FUNCTION_BLOCK FbFiveRung
VAR_INPUT
	xFromSeqLogic: BOOL;
	xEStopOK: BOOL;
	xAutoMode: BOOL;
	xManMode: BOOL;
	xPushButton: BOOL;
	xSensor: BOOL;
	xResetFault: BOOL;
END_VAR
VAR_OUTPUT
	xTrigger: BOOL;
	xSafe: BOOL;
	xCommand: BOOL;
	xInPosition: BOOL;
	xTimeoutFault: BOOL;
END_VAR
VAR
	FaultTimer: TON;
	tETFault: TIME;
END_VAR

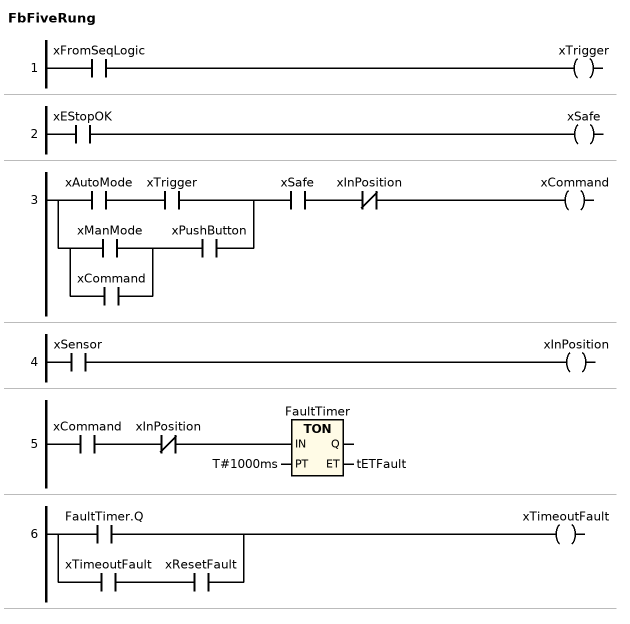
// NETWORK 1
xTrigger := xFromSeqLogic;

// NETWORK 2
xSafe := xEStopOK;

// NETWORK 3
xCommand := (xAutoMode AND xTrigger OR (xManMode OR xCommand) AND xPushButton) AND xSafe AND NOT xInPosition;

// NETWORK 4
xInPosition := xSensor;

// NETWORK 5
FaultTimer(IN := xCommand AND NOT xInPosition, PT := T#1000ms, ET => tETFault); // TON

// NETWORK 6
xTimeoutFault := FaultTimer.Q OR xTimeoutFault AND xResetFault;

END_FUNCTION_BLOCK

(* stored: Version 1.1.0.1, ProductVersion 3.1.4024.12
   POU FbFiveRung: Id {4b06e49f-294b-4ae6-b4fb-f39feaad2da0}, SpecialFunc None *)
